INTERFACE I_HE_SATT_FilterWedge EXTENDS I_HE_SATT_Filter

PROPERTY MaxThickness : LREAL
GET
END_GET
END_PROPERTY

PROPERTY MinThickness : LREAL
GET
END_GET
END_PROPERTY


METHOD ThicknessAt : LREAL
VAR_INPUT
    fPosition : LREAL; // Position in units of property Length and with value from 0 to value of property Length
END_VAR
END_METHOD

END_INTERFACE

(* stored: Version 1.1.0.1
   Itf I_HE_SATT_FilterWedge: Id {07fda710-a856-45c4-9342-2b90967d8a83}
   Property MaxThickness: Id {37b68b46-62a8-4e25-864a-75a9f7bf8336}
   Get Get: Id {a57adced-ca37-4f0a-a390-d0064ce6e00b}
   Property MinThickness: Id {db1d9ef8-484e-41f5-968a-55e08eeada88}
   Get Get: Id {d61d3c84-6847-4fbc-9c71-da60b0c809eb}
   Method ThicknessAt: Id {81688184-8feb-4b22-ab03-0cd1e3659053} *)
